# B&R Automation Studio project Pachore_Mayuresh_Project_3 (part 2)

#### Main.st
```iecst
PROGRAM _INIT
	(* Insert code here *)

END_PROGRAM

PROGRAM _CYCLIC
	(* Insert code here *)

	CASE State OF
		0: //

			IF Service_Mode THEN
				State := 1;
			END_IF

			CASE Crane_Current_State OF

				Crane_Stop_Seq:
					C_Current_State 			:= 'Crane Stop Sequence';
					Start_Crane 				:= FALSE;
					Gantry_Crane.Axis_Command 	:= Emergency_Stop_Req;
					Box_Crane.Axis_Command 		:= Emergency_Stop_Req;
					Crane_Current_State 		:= Crane_Stop_Done;

				Crane_Stop_Done:
					C_Current_State := 'Crane Stop Done';
					IF (Gantry_Crane_Pos_Reached AND Box_Crane_Pos_Reached) THEN
						Gantry_Crane.Axis_Command 	:= Idle;
						Box_Crane.Axis_Command 		:= Idle;
						C_Emergency_Stop 			:= FALSE;
						C_Immediate_Stop 			:= FALSE;
						C_On_Phase_Stop 			:= FALSE;
						Stop_Req 					:= TRUE;
						Crane_Current_State 		:= Wait_Start;
					END_IF

				Reset_Crane_Config:
					C_Current_State := 'Reset Crane Configuration';
					IF NOT C_Reset_Config THEN
						Crane_Current_State := Wait_Start;
					END_IF

					IF (Gantry_Crane_Pos_Reached AND Box_Crane_Pos_Reached AND NOT Box_Holder_Dis_Req AND NOT Pusher_X_En_Req AND NOT Pusher_Z_En_Req AND NOT Vacuum_Dis_Req AND NOT Cartboard_Dis_Req) THEN
						Gantry_Crane.Axis_Command 	:= Idle;
						Box_Crane.Axis_Command 		:= Idle;
						FOR a := 0 TO 9 DO
							En_Dis_Array[a] := FALSE;
						END_FOR;
						C_Reset_Config 		:=FALSE;
						Crane_Current_State := Wait_Start;
					END_IF

				Restore_Crane_Config_1:
					C_Current_State 			:= 'Restore Crane Configuration 1';
					Gantry_Crane.Axis_Command 	:= Idle;
					Box_Crane.Axis_Command 		:= Idle;
					FOR a := 0 TO 9 DO
						IF En_Dis_Array[a] THEN
							CASE a OF
								0:
									Vacuum_En_Req 		:= TRUE;
								1:
									Vacuum_Dis_Req 		:= TRUE;
								2:
									Cartboard_En_Req 	:= TRUE;
								3:
									Cartboard_Dis_Req 	:= TRUE;
								4:
									Box_Holder_En_Req 	:= TRUE;
								5:
									Box_Holder_Dis_Req 	:= TRUE;
								6:
									Pusher_Z_En_Req 	:= TRUE;
								7:
									Pusher_Z_Dis_Req 	:= TRUE;
								8:
									Pusher_X_En_Req 	:= TRUE;
								9:
									Pusher_X_Dis_Req 	:= TRUE;
							END_CASE
						END_IF
					END_FOR
					En_Dis_Counter 		:= 70;
					Crane_Current_State := Restore_Crane_Config_2;

				Restore_Crane_Config_2:
					C_Current_State := 'Restore Crane Configuration 2';
					FOR a := 0 TO 9 DO
						IF En_Dis_Array[a] THEN
							CASE a OF
								0:
									IF NOT Vacuum_En_Req THEN
										En_Dis_Array[a] := FALSE;
									END_IF
								1:
									IF NOT Vacuum_Dis_Req THEN
										En_Dis_Array[a] := FALSE;
									END_IF

								2:
									IF NOT Cartboard_En_Req THEN
										En_Dis_Array[a] := FALSE;
									END_IF

								3:
									IF NOT Cartboard_Dis_Req THEN
										En_Dis_Array[a] := FALSE;
									END_IF

								4:
									IF NOT Box_Holder_En_Req THEN
										En_Dis_Array[a] := FALSE;
									END_IF

								5:
									IF NOT Box_Holder_Dis_Req THEN
										En_Dis_Array[a] := FALSE;
									END_IF

								6:
									IF NOT Pusher_Z_En_Req THEN
										En_Dis_Array[a] := FALSE;
									END_IF

								7:
									IF NOT Pusher_Z_Dis_Req THEN
										En_Dis_Array[a] := FALSE;
									END_IF

								8:
									IF NOT Pusher_X_En_Req THEN
										En_Dis_Array[a] := FALSE;
									END_IF

								9:
									IF NOT Pusher_X_Dis_Req THEN
										En_Dis_Array[a] := FALSE;
									END_IF
							END_CASE
						END_IF
					END_FOR
					En_Dis_Counter := En_Dis_Counter - 1;

					IF En_Dis_Counter = 0 THEN
						IF Check_Pos[0] THEN
							Gantry_Crane_Tar_Pos 		:= Old_Pos[0];
							Gantry_Crane.Axis_Command 	:= Change_Pos;
						END_IF

						IF Check_Pos[1] THEN
							Box_Crane_Tar_Pos 		:= Old_Pos[1];
							Box_Crane.Axis_Command 	:= Change_Pos;
						END_IF
						Crane_Current_State := Restore_Crane_Config_3;
					END_IF

				Restore_Crane_Config_3:
					C_Current_State := 'Restore Crane Configuration 3';
					IF (Gantry_Crane_Pos_Reached AND Check_Pos[0]) THEN
						Gantry_Crane_Pos_Restored := TRUE;
						Gantry_Crane.Axis_Command := Idle;
					END_IF

					IF (Box_Crane_Pos_Reached AND Check_Pos[1]) THEN
						Box_Crane_Pos_Restored := TRUE;
						Box_Crane.Axis_Command := Idle;
					END_IF

					IF (NOT Check_Pos[0] OR Gantry_Crane_Pos_Restored) AND (NOT Check_Pos[1] OR Box_Crane_Pos_Restored) THEN
						Stop_Req 			:= FALSE;
						C_Restart 			:= FALSE;
						Crane_Current_State := Old_State;
					END_IF

				Wait_Start:
					C_Current_State := 'Wait Start';
					IF C_Restart THEN
						Crane_Current_State := Restore_Crane_Config_1;
					END_IF

					IF C_Reset_Config THEN
						Crane_Cartboard_Counter 	:= 28;
						C_Ready						:= FALSE;
						Hold_Boxes 					:= FALSE;
						Load_Boxes_On_The_P 		:= FALSE;
						Boxes_On_The_P 				:= FALSE;
						Box_Holder_Dis_Req 			:= TRUE;
						Pusher_Z_En_Req				:= TRUE;
						Pusher_X_En_Req				:= TRUE;
						Vacuum_Dis_Req 				:= TRUE;
						Cartboard_Dis_Req 			:= TRUE;
						Gantry_Crane_Tar_Pos 		:= 0;
						Gantry_Crane.Axis_Command 	:= Change_Pos;
						Box_Crane_Tar_Pos			:= 0;
						Box_Crane.Axis_Command		:= Change_Pos;
						Crane_Current_State			:= Reset_Crane_Config;
					END_IF

					IF (Start_Crane AND NOT C_Reset_Config AND NOT C_Restart) THEN
						Gantry_Crane_Tar_Pos 		:= 0;
						Gantry_Crane.Axis_Command 	:= Change_Pos;
						Crane_Current_State 		:= Wait_Gantry_Crane_Start_Pos;
					END_IF

					IF C_Emergency_Stop THEN
						Crane_Current_State := Crane_Stop_Seq;
					END_IF

					IF C_Immediate_Stop AND NOT Stop_Req THEN
						Old_State 			:= Crane_Current_State;
						Crane_Current_State := Crane_Stop_Seq;
					END_IF

					IF C_Immediate_Stop AND Stop_Req THEN
						Crane_Current_State := Crane_Stop_Seq;
					END_IF

				Wait_Gantry_Crane_Start_Pos:
					C_Current_State := 'Wait Gantry Crane Start In Position';
					IF (Gantry_Crane_Pos_Reached OR Gantry_Crane_Pos_Restored) THEN
						Check_Pos[0] 				:= FALSE;
						Gantry_Crane_Pos_Restored 	:= FALSE;
						Gantry_Crane.Axis_Command 	:= Idle;
						Box_Crane_Tar_Pos 			:= -0.195;
						Box_Crane.Axis_Command 		:= Change_Pos;
						Crane_Current_State 		:= Wait_Cartboard_Load_Pos;
					END_IF

					IF C_Emergency_Stop THEN
						Crane_Current_State := Crane_Stop_Seq;
					END_IF

					IF C_Immediate_Stop THEN
						Check_Pos[0] 		:= TRUE;
						Old_Pos[0] 			:= 0;
						Old_State 			:= Crane_Current_State;
						Crane_Current_State := Crane_Stop_Seq;
					END_IF

				Wait_Cartboard_Load_Pos:
					C_Current_State := 'Wait Cardboard Load In Position';
					IF (Box_Crane_Pos_Reached OR Box_Crane_Pos_Restored) THEN
						Check_Pos[1] 			:= FALSE;
						Box_Crane_Pos_Restored 	:= FALSE;
						Box_Crane.Axis_Command 	:= Idle;
						Vacuum_En_Req 			:= TRUE;
						Cartboard_En_Req 		:= TRUE;
						Crane_Current_State 	:= Wait_Cartboard_Load;
					END_IF

					IF C_Emergency_Stop THEN
						Crane_Current_State := Crane_Stop_Seq;
					END_IF

					IF C_Immediate_Stop THEN
						Check_Pos[1] 		:= TRUE;
						Old_Pos[1] 			:= -0.195;
						Old_State 			:= Crane_Current_State;
						Crane_Current_State := Crane_Stop_Seq;
					END_IF

				Wait_Cartboard_Load:
					C_Current_State := 'Wait Cardboard Load';
					IF (NOT Vacuum_En_Req AND NOT Cartboard_En_Req) THEN
						Box_Crane_Tar_Pos 		:= 0;
						Box_Crane.Axis_Command 	:= Change_Pos;
						Crane_Current_State 	:= Wait_Box_Crane_Start_Pos;
					END_IF

					IF C_Emergency_Stop THEN
						Crane_Current_State := Crane_Stop_Seq;
					END_IF

					IF C_Immediate_Stop THEN
						En_Dis_Array[0] 	:= TRUE;
						En_Dis_Array[2] 	:= TRUE;
						Old_State 			:= Crane_Current_State;
						Crane_Current_State := Crane_Stop_Seq;
					END_IF

				Wait_Box_Crane_Start_Pos:
					C_Current_State := 'Wait Box Crane Start In Position';
					IF (Box_Crane_Pos_Reached OR Box_Crane_Pos_Restored) THEN
						Check_Pos[1] 			:= FALSE;
						Box_Crane_Pos_Restored 	:= FALSE;
						Box_Crane.Axis_Command 	:= Idle;
						Pusher_Z_En_Req 		:= TRUE;
						Crane_Current_State 	:= Wait_Pusher_Z_Start_Pos_Down;
					END_IF

					IF C_Emergency_Stop THEN
						Crane_Current_State := Crane_Stop_Seq;
					END_IF

					IF C_Immediate_Stop THEN
						Check_Pos[1] 		:= TRUE;
						Old_Pos[1] 			:= 0;
						Old_State 			:= Crane_Current_State;
						Crane_Current_State := Crane_Stop_Seq;
					END_IF

				Wait_Pusher_Z_Start_Pos_Down:
					C_Current_State := 'Wait Pusher Z Start In Position Down';
					IF NOT Pusher_Z_En_Req THEN
						Pusher_X_En_Req 	:= TRUE;
						Crane_Current_State := Wait_Pusher_X_Start_Pos_FWD;
					END_IF

					IF C_Emergency_Stop THEN
						Crane_Current_State := Crane_Stop_Seq;
					END_IF

					IF C_Immediate_Stop THEN
						En_Dis_Array[6] 	:= TRUE;
						Old_State 			:= Crane_Current_State;
						Crane_Current_State := Crane_Stop_Seq;
					END_IF

				Wait_Pusher_X_Start_Pos_FWD:
					C_Current_State := 'Wait Pusher X Start In Position Forward';
					IF NOT Pusher_X_En_Req THEN
						Cartboard_Dis_Req 	:= TRUE;
						Crane_Current_State := Lock_Cartboard;
					END_IF

					IF C_Emergency_Stop THEN
						Crane_Current_State := Crane_Stop_Seq;
					END_IF

					IF C_Immediate_Stop THEN
						En_Dis_Array[8] 	:= TRUE;
						Old_State 			:= Crane_Current_State;
						Crane_Current_State := Crane_Stop_Seq;
					END_IF

				Lock_Cartboard:
					C_Current_State := 'Lock Cardboard';
					IF NOT Cartboard_Dis_Req THEN
						Crane_Cartboard_Counter := Crane_Cartboard_Counter - 1;
						C_Ready 				:= TRUE;
						Crane_Current_State 	:= Wait_Boxes;
					END_IF

					IF C_Emergency_Stop THEN
						Crane_Current_State := Crane_Stop_Seq;
					END_IF

					IF C_Immediate_Stop THEN
						En_Dis_Array[3] 	:= TRUE;
						Old_State 			:= Crane_Current_State;
						Crane_Current_State := Crane_Stop_Seq;
					END_IF

				Wait_Boxes:
					C_Current_State := 'Wait Boxes';
					IF Hold_Boxes THEN
						Box_Holder_En_Req 	:= TRUE;
						Crane_Current_State := Wait_SlideRail_Hold;
					END_IF

					IF C_Emergency_Stop THEN
						Crane_Current_State := Crane_Stop_Seq;
					END_IF

					IF C_Immediate_Stop OR C_On_Phase_Stop THEN
						Old_State 			:= Crane_Current_State;
						Crane_Current_State := Crane_Stop_Seq;
					END_IF

				Wait_SlideRail_Hold:
					C_Current_State := 'Wait SlideRail Hold';
					IF NOT Box_Holder_En_Req THEN
						Pusher_Z_Dis_Req 	:= TRUE;
						Crane_Current_State := Wait_Pusher_Z_Push_Pos_Up;
					END_IF

					IF C_Emergency_Stop THEN
						Crane_Current_State := Crane_Stop_Seq;
					END_IF

					IF C_Immediate_Stop THEN
						En_Dis_Array[4] 	:= TRUE;
						Old_State 			:= Crane_Current_State;
						Crane_Current_State := Crane_Stop_Seq;
					END_IF

				Wait_Pusher_Z_Push_Pos_Up:
					C_Current_State := 'Wait Pusher Z Push Position Up';
					IF NOT Pusher_Z_Dis_Req THEN
						Pusher_X_Dis_Req 	:= TRUE;
						Crane_Current_State := Wait_Pusher_X_Push_Pos_BKW;
					END_IF

					IF C_Emergency_Stop THEN
						Crane_Current_State := Crane_Stop_Seq;
					END_IF

					IF C_Immediate_Stop THEN
						En_Dis_Array[7] 	:= TRUE;
						Old_State 			:= Crane_Current_State;
						Crane_Current_State := Crane_Stop_Seq;
					END_IF

				Wait_Pusher_X_Push_Pos_BKW:
					C_Current_State := 'Wait Pusher Z Push Position Backward';
					IF NOT Pusher_X_Dis_Req THEN
						Pusher_Z_En_Req 	:= TRUE;
						Crane_Current_State := Crane_Idle;
					END_IF

					IF C_Emergency_Stop THEN
						Crane_Current_State := Crane_Stop_Seq;
					END_IF

					IF C_Immediate_Stop THEN
						En_Dis_Array[9] 	:= TRUE;
						Old_State 			:= Crane_Current_State;
						Crane_Current_State := Crane_Stop_Seq;
					END_IF

				Crane_Idle:
					C_Current_State := 'Crane Idle';
					IF (Load_Boxes_On_The_P AND NOT Pusher_Z_En_Req) THEN
						Crane_Current_State := Wait_Pusher_Z_Push_Pos_Down;
					END_IF

					IF C_Emergency_Stop THEN
						Crane_Current_State := Crane_Stop_Seq;
					END_IF

					IF C_Immediate_Stop THEN
						En_Dis_Array[6] 	:= TRUE;
						Old_State 			:= Crane_Current_State;
						Crane_Current_State := Crane_Stop_Seq;
					END_IF

				Wait_Pusher_Z_Push_Pos_Down:
					C_Current_State := 'Wait Pusher Z Push Position Down';
					IF NOT Second_Layer THEN
						Box_Crane_Tar_Pos 		:= -0.2;
						Box_Crane.Axis_Command 	:= Change_Pos;
						Crane_Current_State 	:= Wait_Box_Crane_Cartboard_Pos;
					END_IF

					IF Second_Layer THEN
						Box_Crane_Tar_Pos 		:= 0.01;
						Box_Crane.Axis_Command 	:= Change_Pos;
						Crane_Current_State 	:= Wait_Box_Crane_Cartboard_Pos;
					END_IF

					IF C_Emergency_Stop THEN
						Crane_Current_State := Crane_Stop_Seq;
					END_IF

					IF C_Immediate_Stop THEN
						Old_State 			:= Crane_Current_State;
						Crane_Current_State := Crane_Stop_Seq;
					END_IF

				Wait_Box_Crane_Cartboard_Pos:
					C_Current_State := 'Wait Box Crane Cardboard In Position';
					IF (Box_Crane_Pos_Reached OR Box_Crane_Pos_Restored) THEN
						Check_Pos[1] 				:= FALSE;
						Box_Crane_Pos_Restored 		:= FALSE;
						Box_Crane.Axis_Command 		:= Idle;
						Gantry_Crane_Tar_Pos 		:= -1.11;
						Gantry_Crane.Axis_Command 	:= Change_Pos;
						Crane_Current_State 		:= Wait_Gantry_Crane_Cartboard_Pos;
					END_IF

					IF C_Emergency_Stop THEN
						Crane_Current_State := Crane_Stop_Seq;
					END_IF

					IF C_Immediate_Stop THEN
						Check_Pos[1] := TRUE;
						IF NOT Second_Layer THEN
							Old_Pos[1] := -0.2;
						END_IF
						IF Second_Layer THEN
							Old_Pos[1] := 0.01;
						END_IF
						Old_State 			:= Crane_Current_State;
						Crane_Current_State := Crane_Stop_Seq;
					END_IF

				Wait_Gantry_Crane_Cartboard_Pos:
					C_Current_State := 'Wait Gantry Crane Cardboard In Position';
					IF (Gantry_Crane_Pos_Reached OR Gantry_Crane_Pos_Restored) THEN
						Check_Pos[0] 				:= FALSE;
						Gantry_Crane_Pos_Restored 	:= FALSE;
						Gantry_Crane.Axis_Command 	:= Idle;
						Vacuum_Dis_Req 				:= TRUE;
						Crane_Current_State 		:= Place_Cartboard;
					END_IF

					IF C_Emergency_Stop THEN
						Crane_Current_State := Crane_Stop_Seq;
					END_IF

					IF C_Immediate_Stop THEN
						Check_Pos[0] 		:= TRUE;
						Old_Pos[0] 			:= -1.11;
						Old_State 			:= Crane_Current_State;
						Crane_Current_State := Crane_Stop_Seq;
					END_IF

				Place_Cartboard:
					C_Current_State := 'Place Cardboard';
					IF NOT Vacuum_Dis_Req THEN
						Gantry_Crane_Tar_Pos 		:= -1.3;
						Gantry_Crane.Axis_Command 	:= Change_Pos;
						Crane_Current_State 		:= Place_Boxes;
					END_IF

					IF C_Emergency_Stop THEN
						Crane_Current_State := Crane_Stop_Seq;
					END_IF

					IF C_Immediate_Stop THEN
						En_Dis_Array[1] 	:= TRUE;
						Old_State 			:= Crane_Current_State;
						Crane_Current_State := Crane_Stop_Seq;
					END_IF

				Place_Boxes:
					C_Current_State := 'Place Boxes';
					IF (Gantry_Crane_Pos_Reached OR Gantry_Crane_Pos_Restored) THEN
						Check_Pos[0] := FALSE;
						Gantry_Crane_Pos_Restored := FALSE;
						Gantry_Crane.Axis_Command := Idle;
						Box_Holder_Dis_Req := TRUE;
						Crane_Current_State := Open_SlideRail;
					END_IF

					IF C_Emergency_Stop THEN
						Crane_Current_State := Crane_Stop_Seq;
					END_IF

					IF C_Immediate_Stop THEN
						Check_Pos[0] 		:= TRUE;
						Old_Pos[0] 			:= -1.3;
						Old_State 			:= Crane_Current_State;
						Crane_Current_State := Crane_Stop_Seq;
					END_IF

				Open_SlideRail:
					C_Current_State := 'Open SlideRail';
					IF NOT Box_Holder_Dis_Req THEN
						Pusher_X_En_Req 			:= TRUE;
						Gantry_Crane_Tar_Pos 		:= 0;
						Gantry_Crane.Axis_Command 	:= Change_Pos;
						Crane_Current_State 		:= Pusher_FWD;
					END_IF

					IF C_Emergency_Stop THEN
						Crane_Current_State := Crane_Stop_Seq;
					END_IF

					IF C_Immediate_Stop THEN
						En_Dis_Array[5] 	:= TRUE;
						Old_State 			:= Crane_Current_State;
						Crane_Current_State := Crane_Stop_Seq;
					END_IF

				Pusher_FWD:
					C_Current_State := 'Pusher Forward';
					IF (NOT Pusher_X_En_Req AND (Gantry_Crane_Pos_Reached OR Gantry_Crane_Pos_Restored)) THEN
						Check_Pos[0] 				:= FALSE;
						Gantry_Crane_Pos_Restored 	:= FALSE;
						Gantry_Crane.Axis_Command 	:= Idle;
						Boxes_On_The_P 				:= TRUE;
						Crane_Current_State 		:= Wait_Start;
					END_IF

					IF C_Emergency_Stop THEN
						Crane_Current_State := Crane_Stop_Seq;
					END_IF

					IF C_Immediate_Stop THEN
						En_Dis_Array[8] 	:= TRUE;
						Check_Pos[0] 		:= TRUE;
						Old_Pos[0] 			:= 0;
						Old_State 			:= Crane_Current_State;
						Crane_Current_State := Crane_Stop_Seq;
					END_IF

			END_CASE

			Gantry_Crane(	Axis_Act_Position 	:= I_Gantry_Crane_Act_Pos,
							New_Set_Point 		:= Gantry_Crane_Tar_Pos,
							Axis_Dev_Timer 		:= 400,
							Axis_TGT_Sensor 	:= TRUE);
			O_Gantry_Crane_Tar_Pos 		:= Gantry_Crane.Axis_TGT_Position;
			Gantry_Crane_Pos_Reached 	:= Gantry_Crane.Axis_In_Pos;
			e_Gantry_Crane_Fault 		:= (*Gantry_Crane.Axis_Dev_Fault OR*) Gantry_Crane_Fault_HMI;

			Box_Crane(	Axis_Act_Position 	:= I_Box_Crane_Act_Pos,
						New_Set_Point 		:= Box_Crane_Tar_Pos,
						Axis_Dev_Timer 		:= 400,
						Axis_TGT_Sensor 	:= TRUE);
			O_Box_Crane_Tar_Pos 	:= Box_Crane.Axis_TGT_Position;
			Box_Crane_Pos_Reached 	:= Box_Crane.Axis_In_Pos;
			e_Box_Crane_Fault 		:= (*Box_Crane.Axis_Dev_Fault OR*) Box_Crane_Fault_HMI;

			Cartboard(	Dev_Operation 		:= Operation_Type,
						Dev_Type 			:= Dev_Without_Feedback OR Dev_With_Single_Actuation,
						Dev_Clock 			:= TRUE,
						Dev_Enable_Time 	:= Cartboard_En_Time,
						Dev_Disable_Time 	:= Cartboard_Dis_Time,
						Dev_Diagnose_Enable := TRUE,
						Dev_Enable_Preset 	:= FALSE,
						Dev_Enable_Request 	:= Cartboard_En_Req,
						Dev_Disable_Request := Cartboard_Dis_Req);
			O_Cartboard_Trig 	:= Cartboard.Dev_Enabled;
			e_Cartboard_Fault 	:= (*Cartboard.Dev_Actuator_Fault OR*) Cartboard_Fault_HMI;

			Vacuum(	Dev_Operation 		:= Operation_Type,
					Dev_Type 			:= Dev_With_Enable_Feedback OR Dev_With_Single_Actuation,
					Dev_Enabled_Sensor 	:= I_Vacuum_retention_act,
					Dev_Clock 			:= TRUE,
					Dev_Enable_Time 	:= Vacuum_En_Time,
					Dev_Disable_Time 	:= Vacuum_Dis_Time,
					Dev_Diagnose_Enable := TRUE,
					Dev_Enable_Preset 	:= FALSE,
					Dev_Enable_Request 	:= Vacuum_En_Req,
					Dev_Disable_Request := Vacuum_Dis_Req);
			O_Vacuum_Grip_act 	:= Vacuum.Dev_Enabled;
			e_Vacuum_Fault 		:= (*Vacuum.Dev_Actuator_Fault OR Vacuum.Dev_Enabled_Sensor_Fault OR*) Vacuum_Fault_HMI;

			Box_Holder(	Dev_Operation 		:= Operation_Type,
						Dev_Type 			:= Dev_Without_Feedback OR Dev_With_Single_Actuation,
						Dev_Clock 			:= TRUE,
						Dev_Enable_Time 	:= Box_Holder_En_Time,
						Dev_Disable_Time 	:= Box_Holder_Dis_Time,
						Dev_Diagnose_Enable := TRUE,
						Dev_Enable_Preset 	:= FALSE,
						Dev_Enable_Request 	:= Box_Holder_En_Req,
						Dev_Disable_Request := Box_Holder_Dis_Req);
			O_Box_Holder := Box_Holder.Dev_Enabled;
			e_Box_Holder_Fault 	:= (*Box_Holder.Dev_Actuator_Fault OR*) Box_Holder_Fault_HMI;

			Pusher_X(	Dev_Operation 		:= Operation_Type,
						Dev_Type 			:= Dev_Without_Feedback OR Dev_With_Single_Actuation,
						Dev_Clock 			:= TRUE,
						Dev_Enable_Time 	:= Pusher_X_En_Time,
						Dev_Disable_Time 	:= Pusher_X_Dis_Time,
						Dev_Diagnose_Enable := TRUE,
						Dev_Enable_Preset 	:= FALSE,
						Dev_Enable_Request 	:= Pusher_X_En_Req,
						Dev_Disable_Request := Pusher_X_Dis_Req);
			O_Pusher_x 				:= Pusher_X.Dev_Enabled;
			e_Crane_Pusher_x_Fault 	:= (*Pusher_X.Dev_Actuator_Fault OR*) Crane_Pusher_X_Fault_HMI;

			Pusher_Z(	Dev_Operation 		:= Operation_Type,
						Dev_Type 			:= Dev_Without_Feedback OR Dev_With_Single_Actuation,
						Dev_Clock 			:= TRUE,
						Dev_Enable_Time 	:= Pusher_Z_En_Time,
						Dev_Disable_Time 	:= Pusher_Z_Dis_Time,
						Dev_Diagnose_Enable := TRUE,
						Dev_Enable_Preset 	:= FALSE,
						Dev_Enable_Request 	:= Pusher_Z_En_Req,
						Dev_Disable_Request := Pusher_Z_Dis_Req);
			O_Pusher_z 				:= Pusher_Z.Dev_Enabled;
			e_Crane_Pusher_z_Fault	:= (*Pusher_Z.Dev_Actuator_Fault OR*) Crane_Pusher_Z_Fault_HMI;

		1: //Service Mode
		//Actuation Servicing
			IF NOT Service_Mode THEN
				State := 0;
			END_IF

			O_Vacuum_Grip_act 	:= vaccume_box_crane_grip_HMI;
			O_Cartboard_Trig 	:= Cartboard_Trig_HMI;
			O_Box_Holder := Slide_rail_right_EN_HMI;
			O_Pusher_z 			:= pusher_z_EN_HMI;
			O_Pusher_x 			:= pusher_x_EN_HMI;

			IF gantry_crane_Origin_pos_HMI THEN
				O_Gantry_Crane_Tar_Pos 	:= 0;
			ELSIF gantry_crane_TGT_pos_HMI THEN
				O_Gantry_Crane_Tar_Pos 	:= gantry_crane_TGT_HMI;
			END_IF
			gantry_crane_TGT_dis_HMI 	:= gantry_crane_TGT_HMI;

			IF box_crane_Origin_pos_HMI THEN
				O_Box_Crane_Tar_Pos := 0;
			ELSIF box_crane_TGT_pos_HMI THEN
				O_Box_Crane_Tar_Pos := box_crane_TGT_HMI;
			END_IF
			box_crane_TGT_dis_HMI 	:= box_crane_TGT_HMI;

			vaccume_box_crane_state_HMI := I_Vacuum_retention_act;
			gantry_crane_Act_Pos_HMI 	:= I_Gantry_Crane_Act_Pos;
			box_crane_Act_Pos_HMI 		:= I_Box_Crane_Act_Pos;

	END_CASE

END_PROGRAM

PROGRAM _EXIT
	(* Insert code here *)

END_PROGRAM
```

### Program Logical/Pallet (IEC)

#### Types.typ
```iecst
TYPE
	Pallet_State :
		(
		Pallet_Stop_Seq := 1,
		Pallet_Stop_Done := 2,
		Reset_Pallet_Config_1 := 3,
		Reset_Pallet_Config_2 := 4,
		Reset_Pallet_Config_3 := 5,
		Restore_Pallet_Config_1 := 6,
		Restore_Pallet_Config_2 := 7,
		Restore_Pallet_Config_3 := 8,
		Wait_Start := 9,
		Wait_Lifter_Down := 10,
		Pallet_Fork_Open := 11,
		Wait_Lifter_Up := 12,
		Pallet_Fork_Close := 13,
		Wait_Lifter_Idle := 14,
		Wait_Pallet_Conv_1_Moving := 15,
		Wait_Pallet_Conv_2_Moving := 16,
		Wait_Pallet_Light_Barrier_2 := 17,
		Wait_Stop_Pallet_Conv_1 := 18,
		Wait_Conv_2_Slow_Down := 19,
		Wait_Pallet_Light_Barrier_1 := 20,
		Wait_Stop_Pallet_Conv_2 := 21,
		Wait_Boxes := 22,
		Wait_Restart_Conv_2 := 23,
		Wait_NOT_Pallet_Light_Barrier_2 := 24,
		Wait_Exit_Velocity := 25
		);
END_TYPE
```

#### Variables.var
```iecst
VAR
	State : INT := 0;
	Pallet_Current_State : Pallet_State;
END_VAR
(*Pallet_Lifter*)
VAR
	Pallet_Lifter : Gen_Axis;
	Pallet_Lifter_Pos_Reached : BOOL;
	Pallet_Lifter_Tar_Pos : REAL;
END_VAR
(*Pallet_Fork*)
VAR
	Pallet_Fork : Gen_Device;
	Pallet_Fork_En_Time : INT := 80;
	Pallet_Fork_Dis_Time : INT := 80;
END_VAR
(*Pallet Conveyor 1*)
VAR
	Pallet_Conv_1 : Gen_Device;
	Pallet_Conv_1_En_Time : INT := 20;
	Pallet_Conv_1_Dis_Time : INT := 20;
END_VAR
(*Pallet Conveyor 2*)
VAR
	Pallet_Conv_2 : Gen_Axis;
	Pallet_Conv_2_Vel_Reached : BOOL;
	Pallet_Conv_2_Tar_Vel : REAL;
END_VAR
(*Faults*)
VAR
	En_Dis_Array : ARRAY[0..3] OF BOOL := [4(FALSE)];
	a : INT := 0;
	En_Dis_Counter : INT;
	Check_Pos : BOOL := FALSE;
	Old_Pos : REAL;
	Check_Vel : BOOL;
	Old_Vel : REAL;
	Pallet_Lifter_Pos_Restored : BOOL := FALSE;
	Pallet_Conv_2_Vel_Restored : BOOL := FALSE;
	Pallet_On_Conv_2 : BOOL;
	Old_State : Pallet_State;
	Stop_Req : BOOL := FALSE;
END_VAR
VAR CONSTANT
	Idle : WORD := 0;
	Change_Vel : WORD := 1;
	Change_Pos : WORD := 2;
	Emergency_Stop_Req : WORD := 3;
END_VAR
VAR
	P_Fork_En_Req : BOOL;
	P_Fork_Dis_Req : BOOL;
	P_Conv_1_En_Req : BOOL;
	P_Conv_1_Dis_Req : BOOL;
	New_Variable : USINT;
END_VAR
```

#### Main.st
```iecst
PROGRAM _INIT
	(* Insert code here *)

END_PROGRAM

PROGRAM _CYCLIC
	(* Insert code here *)

	CASE State OF
		0://
			IF Service_Mode THEN
				State := 1;
			END_IF

			CASE Pallet_Current_State OF
				Pallet_Stop_Seq:
					P_Current_State 			:= 'Pallet Stop Sequence';
					Start_Pallet 				:= FALSE;
					P_Conv_1_Dis_Req 			:= TRUE;
					Pallet_Lifter.Axis_Command 	:= Emergency_Stop_Req;
					Pallet_Conv_2.Axis_Command 	:= Emergency_Stop_Req;
					Pallet_Current_State 		:= Pallet_Stop_Done;

				Pallet_Stop_Done:
					P_Current_State := 'Pallet Stop Done';
					IF (NOT P_Conv_1_Dis_Req AND Pallet_Lifter_Pos_Reached AND Pallet_Conv_2_Vel_Reached) THEN
						Pallet_Lifter.Axis_Command 	:= Idle;
						Pallet_Conv_2.Axis_Command 	:= Idle;
						P_Emergency_Stop 			:= FALSE;
						P_Immediate_Stop 			:= FALSE;
						P_On_Phase_Stop 			:= FALSE;
						Stop_Req 					:= TRUE;
						Pallet_Current_State 		:= Wait_Start;
					END_IF

				Reset_Pallet_Config_1:
					P_Current_State := 'Reset Pallet Configuration 1';
					IF NOT P_Reset_Config THEN
						Pallet_Current_State := Wait_Start;
					END_IF

					IF Pallet_Lifter_Pos_Reached THEN
						Pallet_Lifter.Axis_Command 	:= Idle;
						P_Fork_Dis_Req 				:= TRUE;
						Pallet_Current_State 		:= Reset_Pallet_Config_2;
					END_IF

				Reset_Pallet_Config_2:
					P_Current_State := 'Reset Pallet Configuration 2';
					IF NOT P_Fork_Dis_Req THEN
						Pallet_Lifter_Tar_Pos 		:= 0;
						Pallet_Lifter.Axis_Command 	:= Change_Pos;
						Pallet_Current_State 		:= Reset_Pallet_Config_3;
					END_IF

				Reset_Pallet_Config_3:
					P_Current_State := 'Reset Pallet Configuration 3';
					IF Pallet_Lifter_Pos_Reached THEN
						Pallet_Lifter.Axis_Command := Idle;
						FOR a := 0 TO 3 DO
							En_Dis_Array[a] 	:= FALSE;
						END_FOR
						P_Reset_Config 			:= FALSE;
						Pallet_Current_State 	:= Wait_Start;
					END_IF

				Restore_Pallet_Config_1:
					P_Current_State 			:= 'Restore Pallet Configuration 1';
					Pallet_Lifter.Axis_Command 	:= Idle;
					Pallet_Conv_2.Axis_Command 	:= Idle;
					FOR a := 0 TO 3 DO
						IF En_Dis_Array[a] THEN
							CASE a OF
								0:
									P_Fork_En_Req 		:= TRUE;
								1:
									P_Fork_Dis_Req 		:= TRUE;
								2:
									P_Conv_1_En_Req 	:= TRUE;
								3:
									P_Conv_1_Dis_Req 	:= TRUE;
							END_CASE
						END_IF
					END_FOR
					En_Dis_Counter 			:= 70;
					Pallet_Current_State 	:= Restore_Pallet_Config_2;

				Restore_Pallet_Config_2:
					P_Current_State := 'Restore Pallet Configuration 2';
					FOR a := 0 TO 3 DO
						IF En_Dis_Array[a] THEN
							CASE a OF
								0:
									IF NOT P_Fork_En_Req THEN
										En_Dis_Array[a] 	:= FALSE;
									END_IF

								1:
									IF NOT P_Fork_Dis_Req THEN
										En_Dis_Array[a] 	:= FALSE;
									END_IF

								2:
									IF NOT P_Conv_1_En_Req THEN
										En_Dis_Array[a] 	:= FALSE;
									END_IF

								3:
									IF NOT P_Conv_1_Dis_Req THEN
										En_Dis_Array[a] 	:= FALSE;
									END_IF
							END_CASE
						END_IF
					END_FOR
					En_Dis_Counter := En_Dis_Counter - 1;

					IF En_Dis_Counter = 0 THEN
						IF Check_Pos THEN
							Pallet_Lifter_Tar_Pos 		:= Old_Pos;
							Pallet_Lifter.Axis_Command 	:= Change_Pos;
						END_IF

						IF Check_Vel THEN
							Pallet_Conv_2_Tar_Vel 		:= Old_Vel;
							Pallet_Conv_2.Axis_Command 	:= Change_Vel;
						END_IF
						Pallet_Current_State := Restore_Pallet_Config_3;
					END_IF

				Restore_Pallet_Config_3:
					P_Current_State := 'Restore Pallet Configuration 3';
					IF (Pallet_Lifter_Pos_Reached AND Check_Pos) THEN
						Pallet_Lifter_Pos_Restored := TRUE;
						Pallet_Lifter.Axis_Command := Idle;
					END_IF
					IF (Pallet_Conv_2_Vel_Reached AND Check_Vel) THEN
						Pallet_Conv_2_Vel_Restored := TRUE;
						Pallet_Conv_2.Axis_Command := Idle;
					END_IF
					IF (NOT Check_Pos OR Pallet_Lifter_Pos_Reached) AND (NOT Check_Vel OR Pallet_Conv_2_Vel_Reached) THEN
						Stop_Req 				:= FALSE;
						P_Restart 				:= FALSE;
						Pallet_Current_State 	:= Old_State;
					END_IF

				Wait_Start:
					P_Current_State := 'Wait Start';
					IF P_Restart THEN
						Pallet_Current_State := Restore_Pallet_Config_1;
					END_IF

					IF P_Reset_Config THEN
						Pallet_Counter 	:= 5;
						P_Ready 		:= FALSE;
						P_Exit_En 		:= FALSE;
						P_Exit_Done 	:= FALSE;
						IF Pallet_Fork.Dev_Disabled THEN
							Pallet_Lifter_Tar_Pos 		:= 0;
							Pallet_Lifter.Axis_Command 	:= Change_Pos;
							Pallet_Current_State 		:= Reset_Pallet_Config_3;
						ELSE
							Pallet_Lifter_Tar_Pos 		:= -0.258;
							Pallet_Lifter.Axis_Command 	:= Change_Pos;
							Pallet_Current_State 		:= Reset_Pallet_Config_1;
						END_IF
					END_IF

					IF (Start_Pallet AND NOT P_Reset_Config AND NOT P_Restart) THEN
						Pallet_Lifter_Tar_Pos 		:= -0.258;
						Pallet_Lifter.Axis_Command 	:= Change_Pos;
						Pallet_Current_State 		:= Wait_Lifter_Down;
					END_IF

					IF P_Emergency_Stop THEN
						Pallet_Current_State := Pallet_Stop_Seq;
					END_IF

					IF P_Immediate_Stop AND NOT Stop_Req THEN
						IF Pallet_On_Conv_2 THEN
							Check_Vel 			:= TRUE;
							Old_Vel 			:= 0.3;
							Pallet_On_Conv_2 	:= FALSE;
						END_IF
						Old_State 				:= Pallet_Current_State;
						Pallet_Current_State 	:= Pallet_Stop_Seq;
					END_IF

					IF P_Immediate_Stop AND Stop_Req THEN
						Pallet_Current_State := Pallet_Stop_Seq;
					END_IF

				Wait_Lifter_Down:
					P_Current_State := 'Wait Lifter Down';
					IF (Pallet_Lifter_Pos_Reached OR Pallet_Lifter_Pos_Restored) THEN
						Check_Pos 					:= FALSE;
						Pallet_Lifter_Pos_Restored 	:= FALSE;
						Pallet_Lifter.Axis_Command 	:= Idle;
						P_Fork_En_Req 				:= TRUE;
						Pallet_Current_State 		:= Pallet_Fork_Open;
					END_IF

					IF P_Emergency_Stop THEN
						Pallet_Current_State := Pallet_Stop_Seq;
					END_IF

					IF P_Immediate_Stop OR P_On_Phase_Stop THEN
						IF Pallet_On_Conv_2 THEN
							Check_Vel 			:= TRUE;
							Old_Vel 			:= 0.3;
							Pallet_On_Conv_2 	:= FALSE;
						END_IF
						Check_Pos 				:= TRUE;
						Old_Pos 				:= -0.258;
						Old_State 				:= Pallet_Current_State;
						Pallet_Current_State 	:= Pallet_Stop_Seq;
					END_IF

				Pallet_Fork_Open:
					P_Current_State := 'Pallet Fork Open';
					IF NOT P_Fork_En_Req THEN
						Pallet_Lifter_Tar_Pos 		:= -0.12;
						Pallet_Lifter.Axis_Command 	:= Change_Pos;
						Pallet_Current_State 		:= Wait_Lifter_Up;
					END_IF

					IF P_Emergency_Stop THEN
						Pallet_Current_State := Pallet_Stop_Seq;
					END_IF

					IF P_Immediate_Stop THEN
						IF Pallet_On_Conv_2 THEN
							Check_Vel 			:= TRUE;
							Old_Vel 			:= 0.3;
							Pallet_On_Conv_2 	:= FALSE;
						END_IF
						En_Dis_Array[0] 		:= TRUE;
						Old_State 				:= Pallet_Current_State;
						Pallet_Current_State 	:= Pallet_Stop_Seq;
					END_IF

				Wait_Lifter_Up:
					P_Current_State := 'Wait Lifter Up';
					IF (Pallet_Lifter_Pos_Reached OR Pallet_Lifter_Pos_Restored) THEN
						Check_Pos 					:= FALSE;
						Pallet_Lifter_Pos_Restored 	:= FALSE;
						Pallet_Lifter.Axis_Command 	:= Idle;
						P_Fork_Dis_Req 				:= TRUE;
						Pallet_Current_State 		:= Pallet_Fork_Close;
					END_IF

					IF P_Emergency_Stop THEN
						Pallet_Current_State := Pallet_Stop_Seq;
					END_IF

					IF P_Immediate_Stop THEN
						Check_Pos 				:= TRUE;
						Old_Pos 				:= -0.12;
						Old_State 				:= Pallet_Current_State;
						Pallet_Current_State 	:= Pallet_Stop_Seq;
					END_IF

				Pallet_Fork_Close:
					P_Current_State := 'Pallet Fork Close';
					IF NOT P_Fork_Dis_Req THEN
						Pallet_Lifter_Tar_Pos 		:= 0.0;
						Pallet_Lifter.Axis_Command 	:= Change_Pos;
						Pallet_Current_State 		:= Wait_Lifter_Idle;
					END_IF

					IF P_Emergency_Stop THEN
						Pallet_Current_State := Pallet_Stop_Seq;
					END_IF

					IF P_Immediate_Stop THEN
						En_Dis_Array[1] 		:= TRUE;
						Old_State 				:= Pallet_Current_State;
						Pallet_Current_State 	:= Pallet_Stop_Seq;
					END_IF

				Wait_Lifter_Idle:
					P_Current_State := 'Wait Lifter Idle';
					IF (Pallet_Lifter_Pos_Reached OR Pallet_Lifter_Pos_Restored) THEN
						Check_Pos 					:= FALSE;
						Pallet_Lifter_Pos_Restored 	:= FALSE;
						Pallet_Lifter.Axis_Command 	:= Idle;
						Pallet_Counter 				:= Pallet_Counter - 1;
						P_Conv_1_En_Req 			:= TRUE;
						Pallet_Current_State 		:= Wait_Pallet_Conv_1_Moving;
					END_IF

					IF P_Emergency_Stop THEN
						Pallet_Current_State := Pallet_Stop_Seq;
					END_IF

					IF P_Immediate_Stop THEN
						Check_Pos 				:= TRUE;
						Old_Pos 				:= 0.0;
						Old_State 				:= Pallet_Current_State;
						Pallet_Current_State 	:= Pallet_Stop_Seq;
					END_IF

				Wait_Pallet_Conv_1_Moving:
					P_Current_State := 'Wait Pallet Conveyor 1 Moving';
					IF NOT P_Conv_1_En_Req THEN
						Pallet_Conv_2_Tar_Vel 		:= 0.5;
						Pallet_Conv_2.Axis_Command 	:= Change_Vel;
						Pallet_Current_State 		:= Wait_Pallet_Conv_2_Moving;
					END_IF

					IF P_Emergency_Stop THEN
						Pallet_Current_State := Pallet_Stop_Seq;
					END_IF

					IF P_Immediate_Stop THEN
						En_Dis_Array[2] 		:= TRUE;
						Old_State 				:= Pallet_Current_State;
						Pallet_Current_State 	:= Pallet_Stop_Seq;
					END_IF

				Wait_Pallet_Conv_2_Moving:
					P_Current_State := 'Wait Pallet Conveyor 2 Moving';
					IF (Pallet_Conv_2_Vel_Reached OR Pallet_Conv_2_Vel_Restored) THEN
						Check_Vel 					:= FALSE;
						Pallet_Conv_2_Vel_Restored 	:= FALSE;
						Pallet_Conv_2.Axis_Command 	:= Idle;
						Pallet_Current_State 		:= Wait_Pallet_Light_Barrier_2;
					END_IF

					IF P_Emergency_Stop THEN
						Pallet_Current_State := Pallet_Stop_Seq;
					END_IF

					IF P_Immediate_Stop THEN
						En_Dis_Array[2] 		:= TRUE;
						Check_Vel 				:= TRUE;
						Old_Vel 				:= 0.5;
						Old_State 				:= Pallet_Current_State;
						Pallet_Current_State 	:= Pallet_Stop_Seq;
					END_IF

				Wait_Pallet_Light_Barrier_2:
					P_Current_State := 'Wait Pallet Light Barrier 2';
					IF I_IR_Sensor_4 AND (Pallet_Conv_2_Vel_Restored OR NOT Check_Vel) THEN
						Check_Vel 					:= FALSE;
						Pallet_Conv_2_Vel_Restored 	:= FALSE;
						P_Conv_1_Dis_Req 			:= TRUE;
						Pallet_Current_State 		:= Wait_Stop_Pallet_Conv_1;
					END_IF

					IF P_Emergency_Stop THEN
						Pallet_Current_State := Pallet_Stop_Seq;
					END_IF

					IF P_Immediate_Stop THEN
						En_Dis_Array[2] 		:= TRUE;
						Check_Vel 				:= TRUE;
						Old_Vel 				:= 0.5;
						Old_State 				:= Pallet_Current_State;
						Pallet_Current_State 	:= Pallet_Stop_Seq;
					END_IF

				Wait_Stop_Pallet_Conv_1:
					P_Current_State := 'Wait Stop Pallet Conveyor 1';
					IF NOT P_Conv_1_Dis_Req AND (Pallet_Conv_2_Vel_Restored OR NOT Check_Vel) THEN
						Check_Vel 					:= FALSE;
						Pallet_Conv_2_Vel_Restored 	:= FALSE;
						Pallet_Conv_2_Tar_Vel 		:= 0.1;
						Pallet_Conv_2.Axis_Command 	:= Change_Vel;
						Pallet_Current_State 		:= Wait_Conv_2_Slow_Down;
					END_IF

					IF P_Emergency_Stop THEN
						Pallet_Current_State := Pallet_Stop_Seq;
					END_IF

					IF P_Immediate_Stop THEN
						En_Dis_Array[3] 		:= TRUE;
						Check_Vel 				:= TRUE;
						Old_Vel 				:= 0.5;
						Old_State 				:= Pallet_Current_State;
						Pallet_Current_State 	:= Pallet_Stop_Seq;
					END_IF

				Wait_Conv_2_Slow_Down:
					P_Current_State := 'Wait Pallet Conveyor 2 Slow Down';
					IF (Pallet_Conv_2_Vel_Reached OR Pallet_Conv_2_Vel_Restored) THEN
						Check_Vel 					:= FALSE;
						Pallet_Conv_2_Vel_Restored 	:= FALSE;
						Pallet_Conv_2.Axis_Command 	:= Idle;
						Pallet_Current_State 		:= Wait_Pallet_Light_Barrier_1;
					END_IF

					IF P_Emergency_Stop THEN
						Pallet_Current_State := Pallet_Stop_Seq;
					END_IF

					IF P_Immediate_Stop THEN
						En_Dis_Array[3] 		:= TRUE;
						Check_Vel 				:= TRUE;
						Old_Vel 				:= 0.1;
						Old_State 				:= Pallet_Current_State;
						Pallet_Current_State 	:= Pallet_Stop_Seq;
					END_IF

				Wait_Pallet_Light_Barrier_1:
					P_Current_State := 'Wait Pallet Light Barrier 1';
					IF I_IR_Sensor_3 AND (Pallet_Conv_2_Vel_Restored OR NOT Check_Vel) THEN
						Check_Vel 					:= FALSE;
						Pallet_Conv_2_Vel_Restored 	:= FALSE;
						Pallet_Conv_2_Tar_Vel 		:= 0.0;
						Pallet_Conv_2.Axis_Command 	:= Change_Vel;
						Pallet_Current_State 		:= Wait_Stop_Pallet_Conv_2;
					END_IF

					IF P_Emergency_Stop THEN
						Pallet_Current_State := Pallet_Stop_Seq;
					END_IF

					IF P_Immediate_Stop THEN
						Check_Vel 				:= TRUE;
						Old_Vel 				:= 0.1;
						Old_State 				:= Pallet_Current_State;
						Pallet_Current_State 	:= Pallet_Stop_Seq;
					END_IF

				Wait_Stop_Pallet_Conv_2:
					P_Current_State := 'Wait Stop Pallet Conveyor 2';
					IF (Pallet_Conv_2_Vel_Reached OR Pallet_Conv_2_Vel_Restored) THEN
						Check_Vel 					:= FALSE;
						Pallet_Conv_2_Vel_Restored 	:= FALSE;
						Pallet_Conv_2.Axis_Command 	:= Idle;
						P_Ready 					:= TRUE;
						Pallet_Current_State 		:= Wait_Boxes;
					END_IF

					IF P_Emergency_Stop THEN
						Pallet_Current_State := Pallet_Stop_Seq;
					END_IF

					IF P_Immediate_Stop THEN
						Check_Vel 				:= TRUE;
						Old_Vel 				:= 0.0;
						Old_State 				:= Pallet_Current_State;
						Pallet_Current_State 	:= Pallet_Stop_Seq;
					END_IF

				Wait_Boxes:
					P_Current_State := 'Wait Boxes';
					IF P_Exit_En THEN
						Pallet_Conv_2_Tar_Vel 		:= 0.2;
						Pallet_Conv_2.Axis_Command 	:= Change_Vel;
						Pallet_Current_State 		:= Wait_Restart_Conv_2;
					END_IF

					IF P_Emergency_Stop THEN
						Pallet_Current_State := Pallet_Stop_Seq;
					END_IF

					IF P_Immediate_Stop OR P_On_Phase_Stop THEN
						Old_State 				:= Pallet_Current_State;
						Pallet_Current_State 	:= Pallet_Stop_Seq;
					END_IF

				Wait_Restart_Conv_2:
					P_Current_State := 'Wait Pallet Conveyor 2 Restart';
					IF (Pallet_Conv_2_Vel_Reached OR Pallet_Conv_2_Vel_Restored) THEN
						Check_Vel 					:= FALSE;
						Pallet_Conv_2_Vel_Restored 	:= FALSE;
						Pallet_Conv_2.Axis_Command 	:= Idle;
						Pallet_Current_State 		:= Wait_NOT_Pallet_Light_Barrier_2;
					END_IF

					IF P_Emergency_Stop THEN
						Pallet_Current_State := Pallet_Stop_Seq;
					END_IF

					IF P_Immediate_Stop THEN
						Check_Vel 				:= TRUE;
						Old_Vel 				:= 0.2;
						Old_State 				:= Pallet_Current_State;
						Pallet_Current_State 	:= Pallet_Stop_Seq;
					END_IF

				Wait_NOT_Pallet_Light_Barrier_2:
					P_Current_State := 'Wait NOT Pallet Light Barrier 2';
					IF NOT I_IR_Sensor_4 AND (Pallet_Conv_2_Vel_Restored OR NOT Check_Vel) THEN
						Check_Vel 					:= FALSE;
						Pallet_Conv_2_Vel_Restored 	:= FALSE;
						Pallet_Conv_2_Tar_Vel 		:= 0.3;
						Pallet_Conv_2.Axis_Command 	:= Change_Vel;
						Pallet_Current_State 		:= Wait_Exit_Velocity;
					END_IF

					IF P_Emergency_Stop THEN
						Pallet_Current_State := Pallet_Stop_Seq;
					END_IF

					IF P_Immediate_Stop THEN
						Check_Vel 				:= TRUE;
						Old_Vel 				:= 0.2;
						Old_State 				:= Pallet_Current_State;
						Pallet_Current_State 	:= Pallet_Stop_Seq;
					END_IF

				Wait_Exit_Velocity:
					P_Current_State := 'Wait Pallet Conveyor 2 Exit Velocity';
					IF (Pallet_Conv_2_Vel_Reached OR Pallet_Conv_2_Vel_Restored) THEN
						Check_Vel 					:= FALSE;
						Pallet_Conv_2_Vel_Restored 	:= FALSE;
						Pallet_Conv_2.Axis_Command 	:= Idle;
						Pallet_On_Conv_2 			:= TRUE;
						P_Exit_Done 				:= TRUE;
						Pallet_Current_State 		:= Wait_Start;
					END_IF

					IF P_Emergency_Stop THEN
						Pallet_Current_State := Pallet_Stop_Seq;
					END_IF

					IF P_Immediate_Stop THEN
						Check_Vel 				:= TRUE;
						Old_Vel 				:= 0.3;
						Old_State 				:= Pallet_Current_State;
						Pallet_Current_State 	:= Pallet_Stop_Seq;
					END_IF
			END_CASE

			Pallet_Lifter(	Axis_Act_Position 	:= I_Pallet_lift_Act_Pos,
							New_Set_Point 		:= Pallet_Lifter_Tar_Pos,
							Axis_Dev_Timer 		:= 400,
							Axis_TGT_Sensor 	:= TRUE);
			O_Pallet_lift_Tar_Pos 		:= Pallet_Lifter.Axis_TGT_Position;
			Pallet_Lifter_Pos_Reached 	:= Pallet_Lifter.Axis_In_Pos;
			e_Pallet_Lifter_Fault 		:= (*Pallet_Lifter.Axis_Dev_Fault OR*) Pallet_Lifter_Fault_HMI;

			Pallet_Fork(Dev_Operation 		:= Operation_Type,
						Dev_Type 			:= Dev_With_Enable_Feedback OR Dev_With_Single_Actuation,
						Dev_Enabled_Sensor 	:= I_Pallet_holder_State,
						Dev_Clock 			:= TRUE,
						Dev_Enable_Time 	:= Pallet_Fork_En_Time,
						Dev_Disable_Time 	:= Pallet_Fork_Dis_Time,
						Dev_Diagnose_Enable := TRUE,
						Dev_Enable_Preset 	:= FALSE,
						Dev_Enable_Request 	:= P_Fork_En_Req,
						Dev_Disable_Request := P_Fork_Dis_Req);
			O_Pallet_Holder 	:= Pallet_Fork.Dev_Enabled;
			e_Pallet_Fork_Fault := (*Pallet_Fork.Dev_Actuator_Fault OR Pallet_Fork.Dev_Disabled_Sensor_Fault OR *)Pallet_Fork_Fault_HMI;

			Pallet_Conv_1(	Dev_Operation 		:= Operation_Type,
							Dev_Type 			:= Dev_Without_Feedback OR Dev_With_Single_Actuation,
							Dev_Clock 			:= TRUE,
							Dev_Enable_Time 	:= Pallet_Conv_1_En_Time,
							Dev_Disable_Time 	:= Pallet_Conv_1_Dis_Time,
							Dev_Diagnose_Enable := TRUE,
							Dev_Enable_Preset 	:= FALSE,
							Dev_Enable_Request 	:= P_Conv_1_En_Req,
							Dev_Disable_Request := P_Conv_1_Dis_Req);
			O_Conveyor_4 		:= Pallet_Conv_1.Dev_Enabled;
			e_Conveyor_4_Fault 	:= (*Pallet_Conv_1.Dev_Actuator_Fault OR *)Pallet_Conv_1_Fault_HMI;

			Pallet_Conv_2(	Axis_Act_Velocity := O_Conveyor_5_vel,
							New_Set_Point := Pallet_Conv_2_Tar_Vel,
							Axis_Dev_Timer := 400);
			O_Conveyor_5_vel 			:= Pallet_Conv_2.Axis_TGT_Velocity;
			Pallet_Conv_2_Vel_Reached 	:= Pallet_Conv_2.Axis_In_Vel;
			e_Conveyor_5_Fault 			:= (*Pallet_Conv_2.Axis_Dev_Fault OR*) Pallet_Conv_2_Fault_HMI;

		1: //Service Mode
			//Actuation Servicing
			IF NOT Service_Mode THEN
				State := 0;
			END_IF

			O_Pallet_Holder := Pallet_fork_HMI;
			O_Conveyor_4 	:= Conveyor_4_HMI;

				IF NOT O_Conveyor_4 THEN
				O_Conveyor_4 := Conveyor_4_Jog_HMI;
			END_IF

			IF Conveyor_5_S1_HMI THEN
				Conveyor_5_S2_HMI 	:= FALSE;
				O_Conveyor_5_vel 	:= 0.5;
			ELSIF Conveyor_5_S2_HMI THEN
				Conveyor_5_S1_HMI 	:= FALSE;
				O_Conveyor_5_vel 	:= 0.1;
			ELSIF NOT (Conveyor_5_S1_HMI AND Conveyor_5_S2_HMI) THEN
				O_Conveyor_5_vel 	:= 0;
			END_IF

			IF Pallet_Lifter_Origin_pos_HMI THEN
				O_Pallet_lift_Tar_Pos 	:= 0;
			ELSIF Pallet_Lifter_TGT_pos_HMI THEN
				O_Pallet_lift_Tar_Pos 	:= Pallet_Lifter_TGT_HMI;
			END_IF
			Pallet_Lifter_TGT_dis_HMI 	:= Pallet_Lifter_TGT_HMI;

			Pallet_Lifter_Act_Pos_HMI 	:= I_Pallet_lift_Act_Pos;
			Pallet_Holder_State_HMI 	:= I_Pallet_holder_State;
			IR_3_HMI 					:= I_IR_Sensor_3;
			IR_4_HMI 					:= I_IR_Sensor_4;

	END_CASE

END_PROGRAM

PROGRAM _EXIT
	(* Insert code here *)

END_PROGRAM
```

### Program Logical/Signal_Mangement (IEC)

#### Variables.var
```iecst
VAR CONSTANT
	Init : INT := 0;
	Run : INT := 1;
	Start_Config : INT := 2;
	Config : INT := 3;
	Start_Gen : INT := 4;
	Generation : INT := 5;
	Alarm : DINT := 2#0000000000000001;
	Anomaly : DINT := 2#0000000000000010;
	Warning : DINT := 2#0000000000000011;
	Information : DINT := 2#0000000000000100;
	Aux_Reset : DINT := 2#0000001000000000;
	Unconditioned_Reset : DINT := 2#0100000000000000;
	Auto_Conditioned_Reset : DINT := 2#0010000000000000;
	Auto_Provisional_Reset : DINT := 2#0001000000000000;
	Auto_Priority_Reset : DINT := 2#0000100000000000;
	Auto_Reset : DINT := 2#0000010000000000;
	Signal_Type_Mask : DINT := 2#0000000000000111;
END_VAR
(*Message IDs*)
VAR CONSTANT
	m_Turn_Pusher_Fault : INT := 1;
	m_Feeder_Pusher_Fault : INT := 2;
	m_Crane_Pusher_x_Fault : INT := 3;
	m_Crane_Pusher_z_Fault : INT := 4;
	m_Vacuum_Fault : INT := 5;
	m_Pallet_Fork_Fault : INT := 6;
	m_Pallets_Over : INT := 7;
	m_Carriage_Fault : INT := 8;
	m_Gantry_Crane_Fault : INT := 9;
	m_Box_Crane_Fault : INT := 10;
	m_Pallet_Lifter_Fault : INT := 11;
	m_Pallets_Almost_Over : INT := 12;
	m_On_Phase_Stop_Requested : INT := 13;
	m_Emergency_Stop_Requested : INT := 14;
	m_Cartboard_Almost_Over : INT := 15;
	m_Cartboard_Over : INT := 16;
	m_Conveyor_1_Fault : INT := 17;
	m_Conveyor_2_Fault : INT := 18;
	m_Conveyor_3_Fault : INT := 19;
	m_Cartboard_Fault : INT := 20;
	m_Box_Holder_Fault : INT := 21;
	m_Conveyor_4_Fault : INT := 22;
	m_Conveyor_5_Fault : INT := 23;
END_VAR
(*Output IDs*)
VAR CONSTANT
	S_None : DWORD := 16#0000;
	S_Emergency_Stop : DWORD := 16#0001;
	S_Immediate_Stop : DWORD := 16#0002;
	S_On_Phase_Stop : DWORD := 16#0004;
	S_Machine_Out_Of_Phase : DWORD := 16#0100;
	S_Machine_Inhabition : DWORD := 16#0200;
	S_Materials_Run_Out_Lamp : DWORD := 16#0400;
	S_Materials_Run_Out_Buzzer : DWORD := 16#0800;
	S_IO_Diagnostic_Inhabition : DWORD := 16#8000;
END_VAR
VAR
	Signal_Management : Signal_Mng;
	Crane_Temp : BOOL;
	Output_Signals : DWORD;
END_VAR
```

#### Main.st
```iecst
PROGRAM _INIT
	(* Insert code here *)

END_PROGRAM

PROGRAM _CYCLIC
	IF (Operation_Type = Init) THEN
		Signal_Management (Operation_Type 	:= Init);
		Signal_Management (Operation_Type 	:= Start_Config);
		Signal_Management.Operation_Type 	:= Config;
		Operation_Type := Run;
	ELSE
		Signal_Management (Operation_Type 	:= Start_Gen);
		Signal_Management.Operation_Type 	:= Generation;
	END_IF;

	Signal_Management (	Signal_Type 		:= Alarm,
						Signal_Code 		:= m_On_Phase_Stop_Requested,
						Signal_Output 		:= S_On_Phase_Stop,
						Activation_Signal 	:= On_Phase_Stop_HMI);

	Signal_Management (	Signal_Type			:= Alarm OR Aux_Reset,
						Signal_Code 		:= m_Emergency_Stop_Requested,
						Signal_Output 		:= S_Emergency_Stop,
						Activation_Signal 	:= Emergency_Stop_HMI);

	// FEEDER

	// Conveyor 1
	Signal_Management (	Signal_Type 		:= Alarm OR Aux_Reset,
						Signal_Code 		:= m_Conveyor_1_Fault,
						Signal_Output 		:= S_Immediate_Stop,
						Activation_Signal 	:= e_Conveyor_1_Fault);

	// Pusher
	Signal_Management (	Signal_Type 		:= Alarm OR Aux_Reset,
						Signal_Code 		:= m_Feeder_Pusher_Fault,
						Signal_Output 		:= S_Immediate_Stop,
						Activation_Signal 	:= e_Feeder_Pusher_Fault);

	// conveyor 2
	Signal_Management (	Signal_Type 		:= Alarm OR Aux_Reset,
						Signal_Code 		:= m_Conveyor_2_Fault,
						Signal_Output 		:= S_Immediate_Stop,
						Activation_Signal 	:= e_Conveyor_2_Fault);

	// Turnpusher
	Signal_Management (	Signal_Type 		:= Alarm OR Aux_Reset,
						Signal_Code 		:= m_Turn_Pusher_Fault,
						Signal_Output 		:= S_Immediate_Stop,
						Activation_Signal 	:= e_Turn_Pusher_Fault);

	// conveyor 3
	Signal_Management (	Signal_Type 		:= Alarm OR Aux_Reset,
						Signal_Code 		:= m_Conveyor_3_Fault,
						Signal_Output 		:= S_Immediate_Stop,
						Activation_Signal 	:= e_Conveyor_3_Fault);

	// Carriage
	Signal_Management (	Signal_Type 		:= Alarm OR Aux_Reset,
						Signal_Code 		:= m_Carriage_Fault,
						Signal_Output 		:= S_Immediate_Stop,
						Activation_Signal 	:= e_Carriage_Fault);

	// CRANE

	// Box crane
	Signal_Management (	Signal_Type 		:= Alarm OR Aux_Reset,
						Signal_Code 		:= m_Box_Crane_Fault,
						Signal_Output 		:= S_Immediate_Stop,
						Activation_Signal 	:= e_Box_Crane_Fault);

	// Gantry crane
	Signal_Management (	Signal_Type 		:= Alarm OR Aux_Reset,
						Signal_Code 		:= m_Gantry_Crane_Fault,
						Signal_Output 		:= S_Immediate_Stop,
						Activation_Signal 	:= e_Gantry_Crane_Fault);

	// vacuum
	Signal_Management (	Signal_Type 		:= Alarm OR Aux_Reset,
						Signal_Code 		:= m_Vacuum_Fault,
						Signal_Output 		:= S_Immediate_Stop,
						Activation_Signal 	:= e_Vacuum_Fault);

	// cartboard
	Signal_Management (	Signal_Type 		:= Alarm OR Aux_Reset,
						Signal_Code 		:= m_Cartboard_Fault,
						Signal_Output 		:= S_Immediate_Stop,
						Activation_Signal 	:= e_Cartboard_Fault);

	//Pusher X
	Signal_Management (	Signal_Type 		:= Alarm OR Aux_Reset,
						Signal_Code 		:= m_Crane_Pusher_x_Fault,
						Signal_Output 		:= S_Immediate_Stop,
						Activation_Signal 	:= e_Crane_Pusher_x_Fault);

	//pusher Z
	Signal_Management (	Signal_Type 		:= Alarm OR Aux_Reset,
						Signal_Code 		:= m_Crane_Pusher_z_Fault,
						Signal_Output 		:= S_Immediate_Stop,
						Activation_Signal 	:= e_Crane_Pusher_z_Fault);

	// slideRail
	Signal_Management (	Signal_Type 		:= Alarm OR Aux_Reset,
						Signal_Code 		:= m_Box_Holder_Fault,
						Signal_Output 		:= S_Immediate_Stop,
						Activation_Signal 	:= e_Box_Holder_Fault);

	// PALLET

	//Lifter
	Signal_Management (	Signal_Type 		:= Alarm OR Aux_Reset,
						Signal_Code 		:= m_Pallet_Lifter_Fault,
						Signal_Output 		:= S_Immediate_Stop,
						Activation_Signal 	:= e_Pallet_Lifter_Fault);

	// fork
	Signal_Management (	Signal_Type 		:= Alarm OR Aux_Reset,
						Signal_Code 		:= m_Pallet_Fork_Fault,
						Signal_Output 		:= S_Immediate_Stop,
						Activation_Signal 	:= e_Pallet_Fork_Fault);

	//conveyor 1
	Signal_Management (	Signal_Type 		:= Alarm OR Aux_Reset,
						Signal_Code 		:= m_Conveyor_4_Fault,
						Signal_Output 		:= S_Immediate_Stop,
						Activation_Signal 	:= e_Conveyor_4_Fault);

	// conveyor 2
	Signal_Management (	Signal_Type 		:= Alarm OR Aux_Reset,
						Signal_Code 		:= m_Conveyor_5_Fault,
						Signal_Output 		:= S_Immediate_Stop,
						Activation_Signal 	:= e_Conveyor_5_Fault);

	// PALLET ALMOST OVER
	Signal_Management (	Signal_Type 		:= Warning,
						Signal_Code 		:= m_Pallets_Almost_Over,
						Signal_Output 		:= S_Machine_Out_Of_Phase,
						Activation_Signal 	:= (Pallet_Counter = 1));

	// PALLET OVER
	Signal_Management (	Signal_Type 		:= Alarm,
						Signal_Code 		:= m_Pallets_Over,
						Signal_Output 		:= S_On_Phase_Stop,
						Activation_Signal 	:= (Pallet_Counter = 0));

	// CARTBOARD ALMOST OVER
	Signal_Management (	Signal_Type 		:= Warning,
						Signal_Code 		:= m_Cartboard_Almost_Over,
						Signal_Output 		:= S_Materials_Run_Out_Lamp,
						Activation_Signal 	:= (Crane_Cartboard_Counter = 1));

	// CARTBOARD OVER
	Signal_Management (	Signal_Type 		:= Alarm,
						Signal_Code 		:= m_Cartboard_Over,
						Signal_Output 		:= S_On_Phase_Stop,
						Activation_Signal 	:= (Crane_Cartboard_Counter = 0));

	Output_Signals 			:= Signal_Management.Signal_Outputs;

	IF (Operation_Type = Run) THEN
		Signal_Management (Operation_Type := Run); (* outputs selection *)
	END_IF;

	Emergency_Stop 			:= ((Output_Signals AND S_Emergency_Stop) = S_Emergency_Stop);

	IF Emergency_Stop THEN
		Immediate_Stop		:= FALSE;
		On_Phase_Stop		:= FALSE;
	END_IF

	IF NOT Emergency_Stop THEN
		Immediate_Stop 		:= ((Output_Signals AND S_Immediate_Stop) = S_Immediate_Stop);
		On_Phase_Stop		:= FALSE;
		IF NOT Immediate_Stop THEN
			On_Phase_Stop 	:= ((Output_Signals AND S_On_Phase_Stop) = S_On_Phase_Stop);
		END_IF;
	END_IF

	Out_Of_Material		:= ((((Output_Signals AND S_Materials_Run_Out_Lamp) = S_Materials_Run_Out_Lamp)) OR (((Output_Signals AND S_Machine_Out_Of_Phase) = S_Machine_Out_Of_Phase)));

	Priority_1_HMI 		:= Fault[Signal_Management.First_Active_Signal_Index];
	Priority_2_HMI 		:= Fault[Signal_Management.Second_Active_Signal_Index];
	Priority_3_HMI 		:= Fault[Signal_Management.Third_Active_Signal_Index];
	Priority_4_HMI 		:= Fault[Signal_Management.Fourth_Active_Signal_Index];

	Aux_Reset_Unlocked 	:= Signal_Management.Aux_Reset_Enable;
	IF Aux_Reset_Unlocked THEN
		Aux_Unlocked	( LED_State := 'blink');
	ELSIF NOT Aux_Reset_Unlocked THEN
		Aux_Unlocked	( LED_State := 'off');
	END_IF

	Reset_Unlocked 		:= Signal_Management.Reset_Enable;
	IF Reset_Unlocked THEN
		R_Unlocked		( LED_State := 'blink');
	ELSIF NOT Reset_Unlocked THEN
		R_Unlocked		( LED_State := 'off');
	END_IF

	IF Signal_Management.First_Active_Signal_Index > 0 AND NOT (Signal_Management.First_Active_Signal_Index = 12 OR Signal_Management.First_Active_Signal_Index = 13 OR Signal_Management.First_Active_Signal_Index = 14 OR Signal_Management.First_Active_Signal_Index = 15) THEN
		Alarm_Detected( LED_State := 'blink');
	ELSIF Signal_Management.First_Active_Signal_Index > 0 AND (Signal_Management.First_Active_Signal_Index = 12 OR Signal_Management.First_Active_Signal_Index = 15) AND NOT (Signal_Management.First_Active_Signal_Index = 13 OR Signal_Management.First_Active_Signal_Index = 14) THEN
		Warning_Detected( LED_State := 'blink');
	ELSE
		Warning_Detected( LED_State := 'off');
		Alarm_Detected( LED_State := 'off');

	END_IF

END_PROGRAM

PROGRAM _EXIT
	(* Insert code here *)

END_PROGRAM
```

Listed in the project but not available here: Logical/MNG_Global.typ, Logical/Global.typ, Logical/Libraries/ComTCP/ComTCP_L/MNG_InternalTyp.hpp, Logical/Libraries/ComTCP/ComTCP_L/MNG_ComHdlr.cpp, Logical/Libraries/S_filter/Types.typ, Logical/Libraries/S_filter/Constants.var, Logical/Libraries/Signal_Mng/Types.typ, Logical/Libraries/Blink/Types.typ, Logical/Libraries/Blink/Constants.var
